% RSLogix 500 project HotWater_HX_12032008.RSS, saved by version 8.10.00.24 %
PROJECT "B8_HW"    % processor: Bul.1763 MicroLogix 1100 Series A %

PROGRAM FILES
  LAD 2 "MAIN"  10 rungs
  LAD 4 "ANALOG IN"  10 rungs
  LAD 5 "PUMP 3"  17 rungs
  LAD 6 "PUMP 4"  16 rungs
  LAD 7 "PRESS PID"  15 rungs
  LAD 8 "TEMP PID"  16 rungs
  LAD 9 "ANALOG OUT"  8 rungs
  LAD 10 "LCD INFO"  13 rungs

DATA FILES
  O0 OUTPUT  8 elements
  I1 INPUT  22 elements
  S2 STATUS  66 elements
  B3 BINARY  11 elements
  T4 TIMER  57 elements
  C5 COUNTER  10 elements
  R6 CONTROL  1 elements
  N7 INTEGER  100 elements
  F8 FLOAT  1 elements
  PD9   12 elements
  N10   200 elements
  N11   52 elements
  N12   40 elements
  F13   40 elements

LADDER 2 "MAIN"
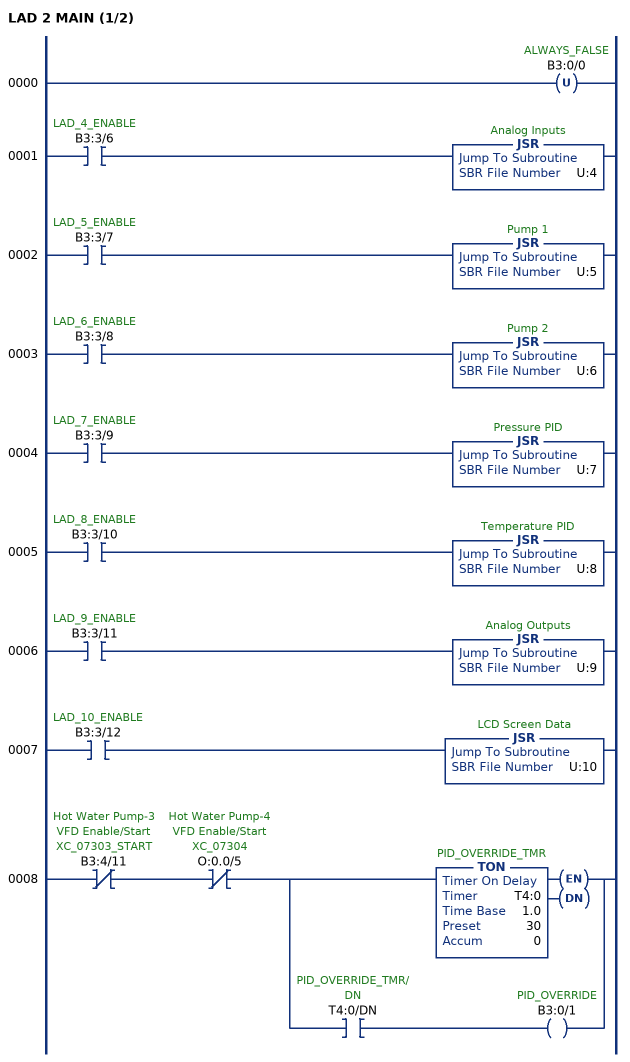
% Rung: 0 %
SOR OTU B3:0/0 EOR
%   B3:0/0  ALWAYS_FALSE %
% Rung: 1 %
SOR XIC B3:3/6 JSR U:4 EOR
%   B3:3/6  LAD_4_ENABLE %
%   U:4  "Analog Inputs" %
% Rung: 2 %
SOR XIC B3:3/7 JSR U:5 EOR
%   B3:3/7  LAD_5_ENABLE %
%   U:5  "Pump 1" %
% Rung: 3 %
SOR XIC B3:3/8 JSR U:6 EOR
%   B3:3/8  LAD_6_ENABLE %
%   U:6  "Pump 2" %
% Rung: 4 %
SOR XIC B3:3/9 JSR U:7 EOR
%   B3:3/9  LAD_7_ENABLE %
%   U:7  "Pressure PID" %
% Rung: 5 %
SOR XIC B3:3/10 JSR U:8 EOR
%   B3:3/10  LAD_8_ENABLE %
%   U:8  "Temperature PID" %
% Rung: 6 %
SOR XIC B3:3/11 JSR U:9 EOR
%   B3:3/11  LAD_9_ENABLE %
%   U:9  "Analog Outputs" %
% Rung: 7 %
SOR XIC B3:3/12 JSR U:10 EOR
%   B3:3/12  LAD_10_ENABLE %
%   U:10  "LCD Screen Data" %
% Rung: 8 %
SOR XIO B3:4/11 XIO O:0.0/5 BST TON T4:0 1.0 30 0 NXB XIC T4:0/DN OTE B3:0/1 BND EOR
%   B3:4/11  XC_07303_START  "Hot Water Pump-3 VFD Enable/Start" %
%   O:0.0/5  XC_07304  "Hot Water Pump-4 VFD Enable/Start" %
%   T4:0  PID_OVERRIDE_TMR %
%   B3:0/1  PID_OVERRIDE %

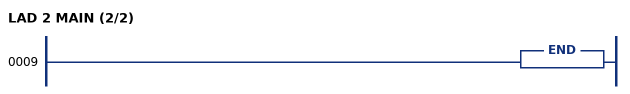
% Rung: 9 %
SOR END EOR

LADDER 4 "ANALOG IN"
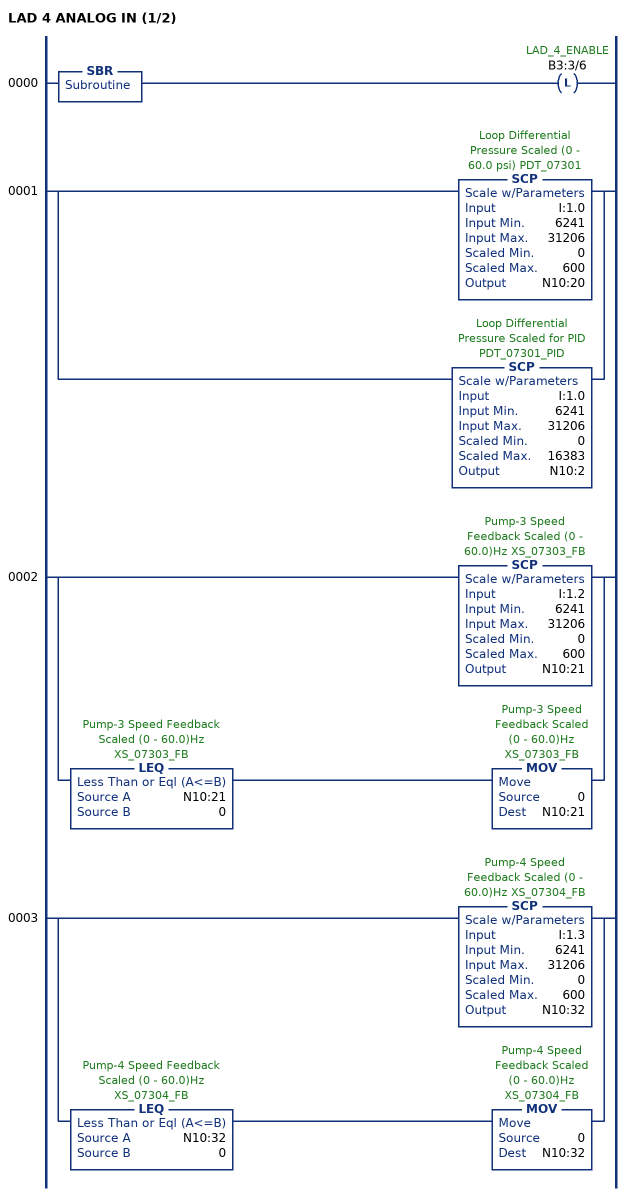
% Rung: 0 %
SOR SBR OTL B3:3/6 EOR
%   B3:3/6  LAD_4_ENABLE %
% Rung: 1 %
SOR BST SCP I:1.0 6241 31206 0 600 N10:20 NXB SCP I:1.0 6241 31206 0 16383 N10:2 BND EOR
%   I:1.0  PDT_07301_RAW  "Loop Differential Pressure Scaled (0.0 - 60.0) psi" %
%   N10:20  PDT_07301  "Loop Differential Pressure Scaled (0 - 60.0 psi)" %
%   N10:2  PDT_07301_PID  "Loop Differential Pressure Scaled for PID" %
% Rung: 2 %
SOR BST SCP I:1.2 6241 31206 0 600 N10:21 NXB LEQ N10:21 0 MOV 0 N10:21 BND EOR
%   I:1.2  XS_07303_FB_RAW  "Pump-3 VFD Speed Feedback" %
%   N10:21  XS_07303_FB  "Pump-3 Speed Feedback Scaled (0 - 60.0)Hz" %
% Rung: 3 %
SOR BST SCP I:1.3 6241 31206 0 600 N10:32 NXB LEQ N10:32 0 MOV 0 N10:32 BND EOR
%   I:1.3  XS_07304_FB_RAW  "Pump-4 VFD Speed Feedback" %
%   N10:32  XS_07304_FB  "Pump-4 Speed Feedback Scaled (0 - 60.0)Hz" %

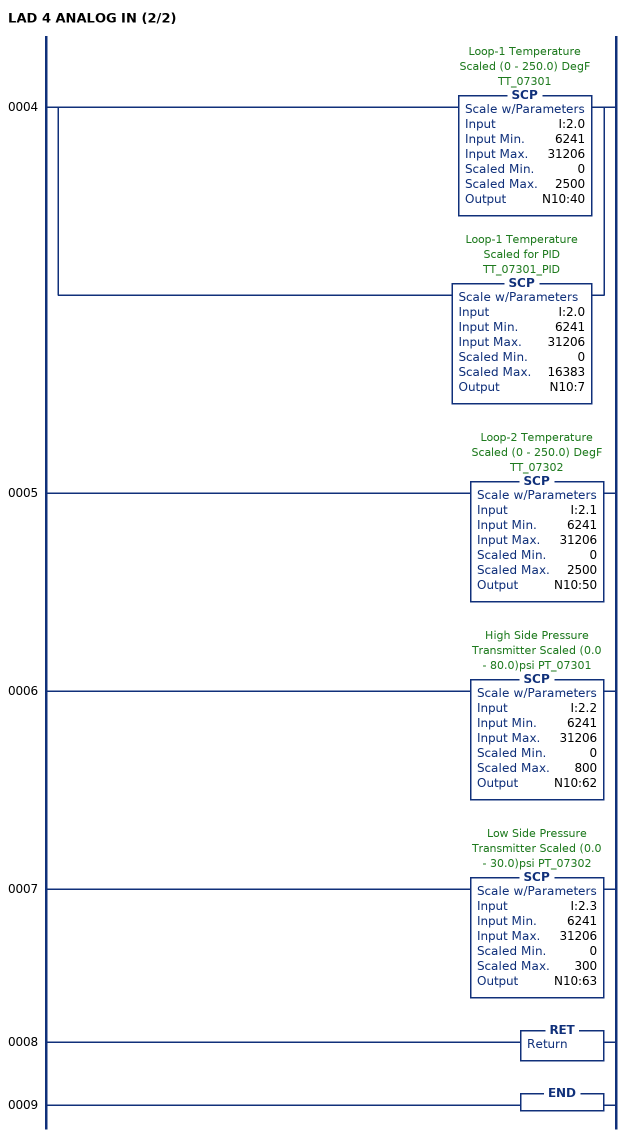
% Rung: 4 %
SOR BST SCP I:2.0 6241 31206 0 2500 N10:40 NXB SCP I:2.0 6241 31206 0 16383 N10:7 BND EOR
%   I:2.0  TT_07301_RAW  "Loop-1 Temperature Transmitter Scaled (0 - 250.0) DegF" %
%   N10:40  TT_07301  "Loop-1 Temperature Scaled (0 - 250.0) DegF" %
%   N10:7  TT_07301_PID  "Loop-1 Temperature Scaled for PID" %
% Rung: 5 %
SOR SCP I:2.1 6241 31206 0 2500 N10:50 EOR
%   I:2.1  TT_07302_RAW  "Loop-2 Temperature Transmitter Scaled (0 - 250.0) DegF" %
%   N10:50  TT_07302  "Loop-2 Temperature Scaled (0 - 250.0) DegF" %
% Rung: 6 %
SOR SCP I:2.2 6241 31206 0 800 N10:62 EOR
%   I:2.2  PT_07301_RAW  "High Side Pressure Transmitter Scaled (0.0 - 80.0)psi" %
%   N10:62  PT_07301  "High Side Pressure Transmitter Scaled (0.0 - 80.0)psi" %
% Rung: 7 %
SOR SCP I:2.3 6241 31206 0 300 N10:63 EOR
%   I:2.3  PT_07302_RAW  "Low Side Pressure Transmitter Scaled (0.0 - 30.0)psi" %
%   N10:63  PT_07302  "Low Side Pressure Transmitter Scaled (0.0 - 30.0)psi" %
% Rung: 8 %
SOR RET EOR
% Rung: 9 %
SOR END EOR

LADDER 5 "PUMP 3"
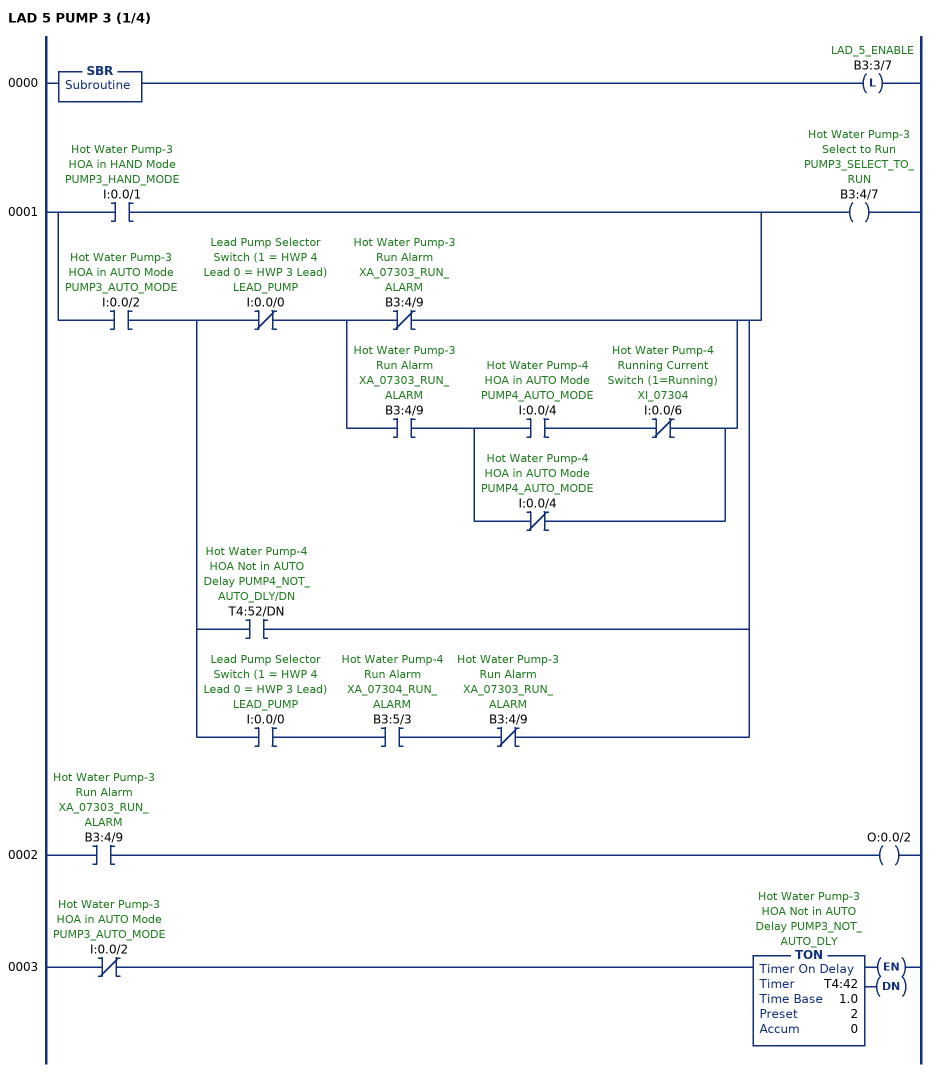
% Rung: 0 %
SOR SBR OTL B3:3/7 EOR
%   B3:3/7  LAD_5_ENABLE %
% Rung: 1 %
SOR BST XIC I:0.0/1 NXB XIC I:0.0/2 BST XIO I:0.0/0 BST XIO B3:4/9 NXB XIC B3:4/9 BST XIC I:0.0/4 XIO I:0.0/6 NXB XIO I:0.0/4 BND BND NXB XIC T4:52/DN NXB XIC I:0.0/0 XIC B3:5/3 XIO B3:4/9 BND BND OTE B3:4/7 EOR
%   I:0.0/1  PUMP3_HAND_MODE  "Hot Water Pump-3 HOA in HAND Mode" %
%   I:0.0/2  PUMP3_AUTO_MODE  "Hot Water Pump-3 HOA in AUTO Mode" %
%   I:0.0/0  LEAD_PUMP  "Lead Pump Selector Switch (1 = HWP 4 Lead 0 = HWP 3 Lead)" %
%   B3:4/9  XA_07303_RUN_ALARM  "Hot Water Pump-3 Run Alarm" %
%   I:0.0/4  PUMP4_AUTO_MODE  "Hot Water Pump-4 HOA in AUTO Mode" %
%   I:0.0/6  XI_07304  "Hot Water Pump-4 Running Current Switch (1=Running)" %
%   T4:52  PUMP4_NOT_AUTO_DLY  "Hot Water Pump-4 HOA Not in AUTO Delay" %
%   B3:5/3  XA_07304_RUN_ALARM  "Hot Water Pump-4 Run Alarm" %
%   B3:4/7  PUMP3_SELECT_TO_RUN  "Hot Water Pump-3 Select to Run" %
% Rung: 2 %
SOR XIC B3:4/9 OTE O:0.0/2 EOR
%   B3:4/9  XA_07303_RUN_ALARM  "Hot Water Pump-3 Run Alarm" %
% Rung: 3 %
SOR XIO I:0.0/2 TON T4:42 1.0 2 0 EOR
%   I:0.0/2  PUMP3_AUTO_MODE  "Hot Water Pump-3 HOA in AUTO Mode" %
%   T4:42  PUMP3_NOT_AUTO_DLY  "Hot Water Pump-3 HOA Not in AUTO Delay" %

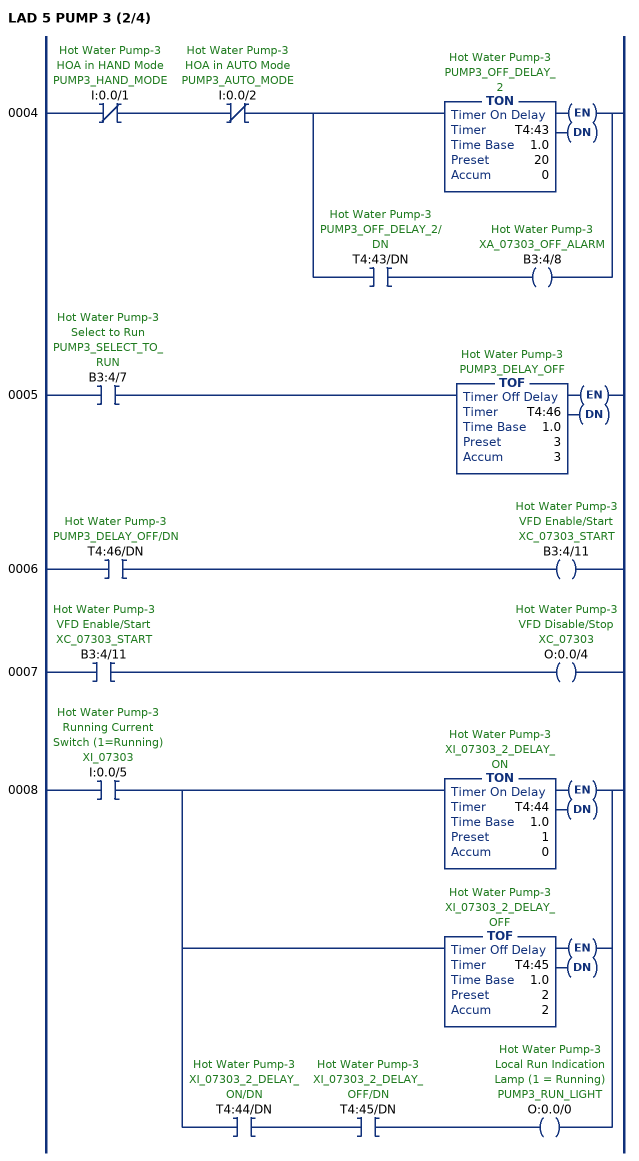
% Rung: 4 %
SOR XIO I:0.0/1 XIO I:0.0/2 BST TON T4:43 1.0 20 0 NXB XIC T4:43/DN OTE B3:4/8 BND EOR
%   I:0.0/1  PUMP3_HAND_MODE  "Hot Water Pump-3 HOA in HAND Mode" %
%   I:0.0/2  PUMP3_AUTO_MODE  "Hot Water Pump-3 HOA in AUTO Mode" %
%   T4:43  PUMP3_OFF_DELAY_2  "Hot Water Pump-3" %
%   B3:4/8  XA_07303_OFF_ALARM  "Hot Water Pump-3" %
% Rung: 5 %
SOR XIC B3:4/7 TOF T4:46 1.0 3 3 EOR
%   B3:4/7  PUMP3_SELECT_TO_RUN  "Hot Water Pump-3 Select to Run" %
%   T4:46  PUMP3_DELAY_OFF  "Hot Water Pump-3" %
% Rung: 6 %
SOR XIC T4:46/DN OTE B3:4/11 EOR
%   T4:46  PUMP3_DELAY_OFF  "Hot Water Pump-3" %
%   B3:4/11  XC_07303_START  "Hot Water Pump-3 VFD Enable/Start" %
% Rung: 7 %
SOR XIC B3:4/11 OTE O:0.0/4 EOR
%   B3:4/11  XC_07303_START  "Hot Water Pump-3 VFD Enable/Start" %
%   O:0.0/4  XC_07303  "Hot Water Pump-3 VFD Disable/Stop" %
% Rung: 8 %
SOR XIC I:0.0/5 BST TON T4:44 1.0 1 0 NXB TOF T4:45 1.0 2 2 NXB XIC T4:44/DN XIC T4:45/DN OTE O:0.0/0 BND EOR
%   I:0.0/5  XI_07303  "Hot Water Pump-3 Running Current Switch (1=Running)" %
%   T4:44  XI_07303_2_DELAY_ON  "Hot Water Pump-3" %
%   T4:45  XI_07303_2_DELAY_OFF  "Hot Water Pump-3" %
%   O:0.0/0  PUMP3_RUN_LIGHT  "Hot Water Pump-3 Local Run Indication Lamp (1 = Running)" %

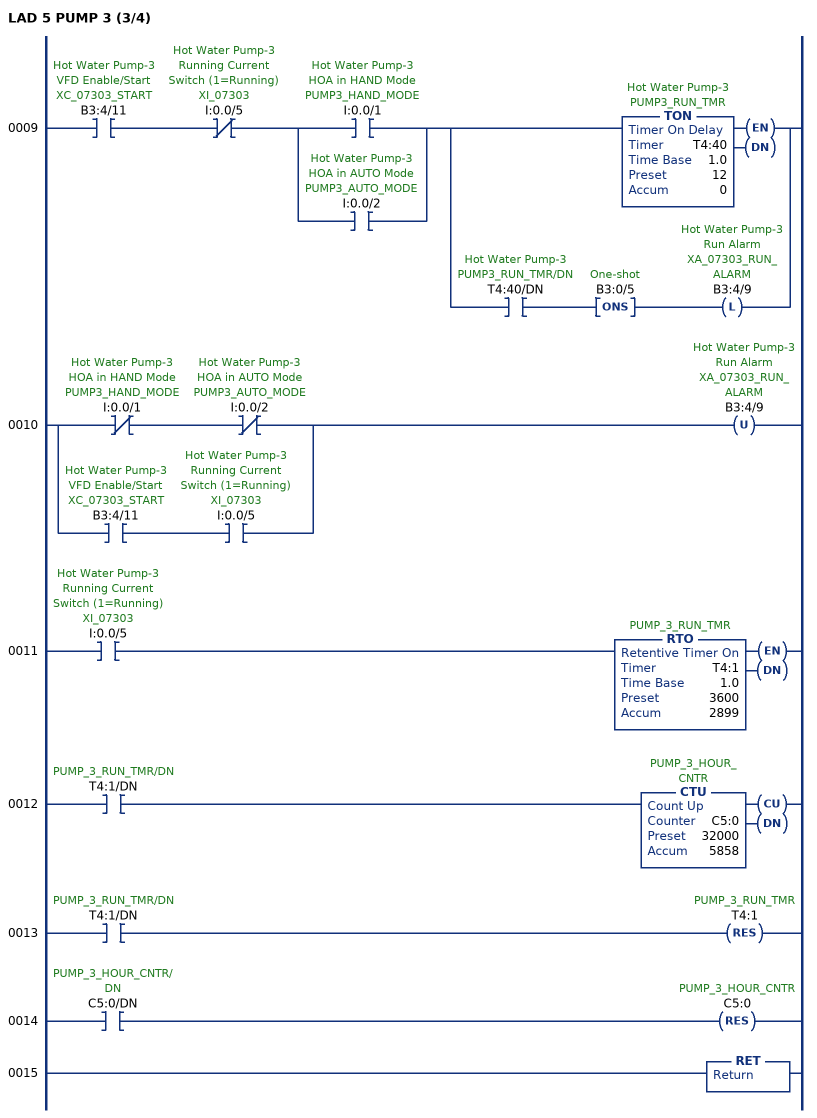
% Rung: 9 %
SOR XIC B3:4/11 XIO I:0.0/5 BST XIC I:0.0/1 NXB XIC I:0.0/2 BND BST TON T4:40 1.0 12 0 NXB XIC T4:40/DN ONS B3:0/5 OTL B3:4/9 BND EOR
%   B3:4/11  XC_07303_START  "Hot Water Pump-3 VFD Enable/Start" %
%   I:0.0/5  XI_07303  "Hot Water Pump-3 Running Current Switch (1=Running)" %
%   I:0.0/1  PUMP3_HAND_MODE  "Hot Water Pump-3 HOA in HAND Mode" %
%   I:0.0/2  PUMP3_AUTO_MODE  "Hot Water Pump-3 HOA in AUTO Mode" %
%   T4:40  PUMP3_RUN_TMR  "Hot Water Pump-3" %
%   B3:0/5  "One-shot" %
%   B3:4/9  XA_07303_RUN_ALARM  "Hot Water Pump-3 Run Alarm" %
% Rung: 10 %
SOR BST XIO I:0.0/1 XIO I:0.0/2 NXB XIC B3:4/11 XIC I:0.0/5 BND OTU B3:4/9 EOR
%   I:0.0/1  PUMP3_HAND_MODE  "Hot Water Pump-3 HOA in HAND Mode" %
%   I:0.0/2  PUMP3_AUTO_MODE  "Hot Water Pump-3 HOA in AUTO Mode" %
%   B3:4/11  XC_07303_START  "Hot Water Pump-3 VFD Enable/Start" %
%   I:0.0/5  XI_07303  "Hot Water Pump-3 Running Current Switch (1=Running)" %
%   B3:4/9  XA_07303_RUN_ALARM  "Hot Water Pump-3 Run Alarm" %
% Rung: 11 %
SOR XIC I:0.0/5 RTO T4:1 1.0 3600 2899 EOR
%   I:0.0/5  XI_07303  "Hot Water Pump-3 Running Current Switch (1=Running)" %
%   T4:1  PUMP_3_RUN_TMR %
% Rung: 12 %
SOR XIC T4:1/DN CTU C5:0 32000 5858 EOR
%   T4:1  PUMP_3_RUN_TMR %
%   C5:0  PUMP_3_HOUR_CNTR %
% Rung: 13 %
SOR XIC T4:1/DN RES T4:1 EOR
%   T4:1  PUMP_3_RUN_TMR %
% Rung: 14 %
SOR XIC C5:0/DN RES C5:0 EOR
%   C5:0  PUMP_3_HOUR_CNTR %
% Rung: 15 %
SOR RET EOR

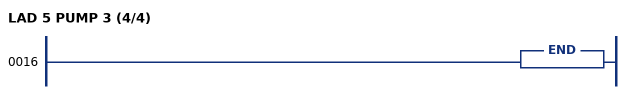
% Rung: 16 %
SOR END EOR

LADDER 6 "PUMP 4"
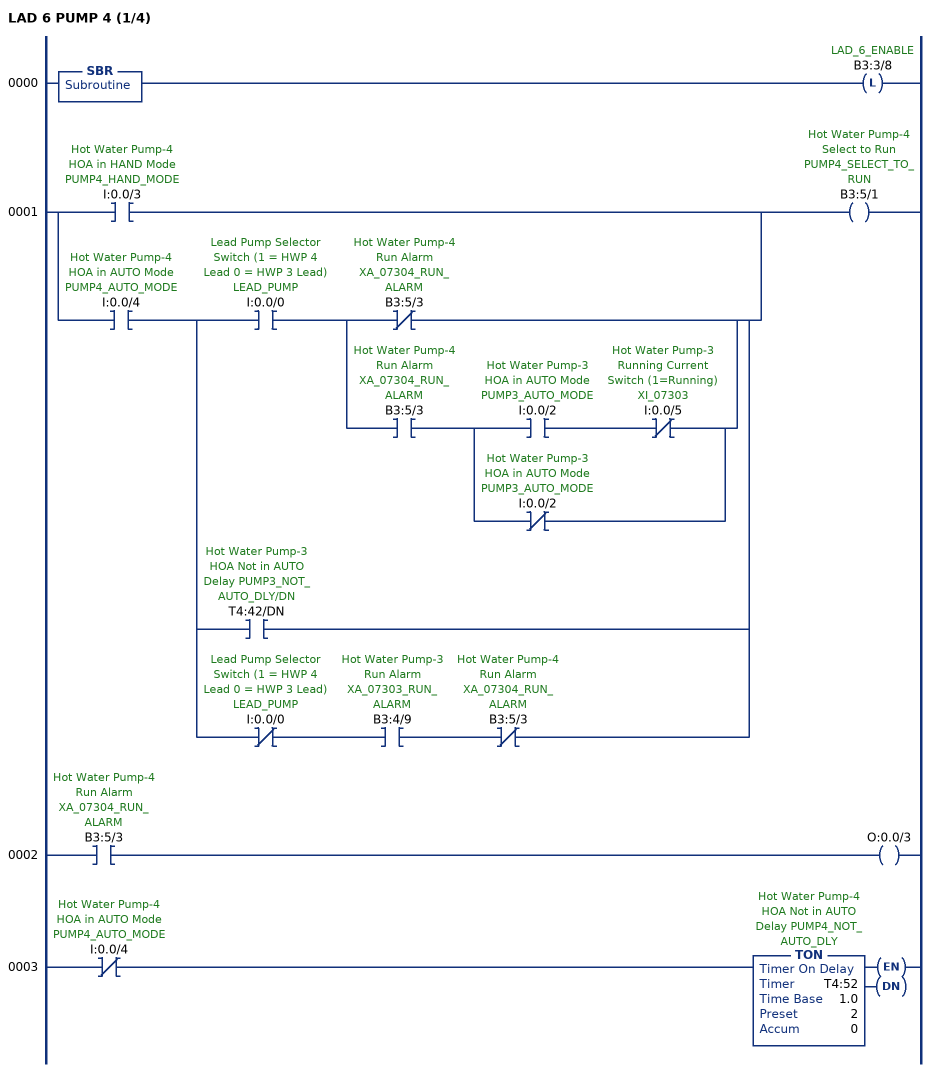
% Rung: 0 %
SOR SBR OTL B3:3/8 EOR
%   B3:3/8  LAD_6_ENABLE %
% Rung: 1 %
SOR BST XIC I:0.0/3 NXB XIC I:0.0/4 BST XIC I:0.0/0 BST XIO B3:5/3 NXB XIC B3:5/3 BST XIC I:0.0/2 XIO I:0.0/5 NXB XIO I:0.0/2 BND BND NXB XIC T4:42/DN NXB XIO I:0.0/0 XIC B3:4/9 XIO B3:5/3 BND BND OTE B3:5/1 EOR
%   I:0.0/3  PUMP4_HAND_MODE  "Hot Water Pump-4 HOA in HAND Mode" %
%   I:0.0/4  PUMP4_AUTO_MODE  "Hot Water Pump-4 HOA in AUTO Mode" %
%   I:0.0/0  LEAD_PUMP  "Lead Pump Selector Switch (1 = HWP 4 Lead 0 = HWP 3 Lead)" %
%   B3:5/3  XA_07304_RUN_ALARM  "Hot Water Pump-4 Run Alarm" %
%   I:0.0/2  PUMP3_AUTO_MODE  "Hot Water Pump-3 HOA in AUTO Mode" %
%   I:0.0/5  XI_07303  "Hot Water Pump-3 Running Current Switch (1=Running)" %
%   T4:42  PUMP3_NOT_AUTO_DLY  "Hot Water Pump-3 HOA Not in AUTO Delay" %
%   B3:4/9  XA_07303_RUN_ALARM  "Hot Water Pump-3 Run Alarm" %
%   B3:5/1  PUMP4_SELECT_TO_RUN  "Hot Water Pump-4 Select to Run" %
% Rung: 2 %
SOR XIC B3:5/3 OTE O:0.0/3 EOR
%   B3:5/3  XA_07304_RUN_ALARM  "Hot Water Pump-4 Run Alarm" %
% Rung: 3 %
SOR XIO I:0.0/4 TON T4:52 1.0 2 0 EOR
%   I:0.0/4  PUMP4_AUTO_MODE  "Hot Water Pump-4 HOA in AUTO Mode" %
%   T4:52  PUMP4_NOT_AUTO_DLY  "Hot Water Pump-4 HOA Not in AUTO Delay" %

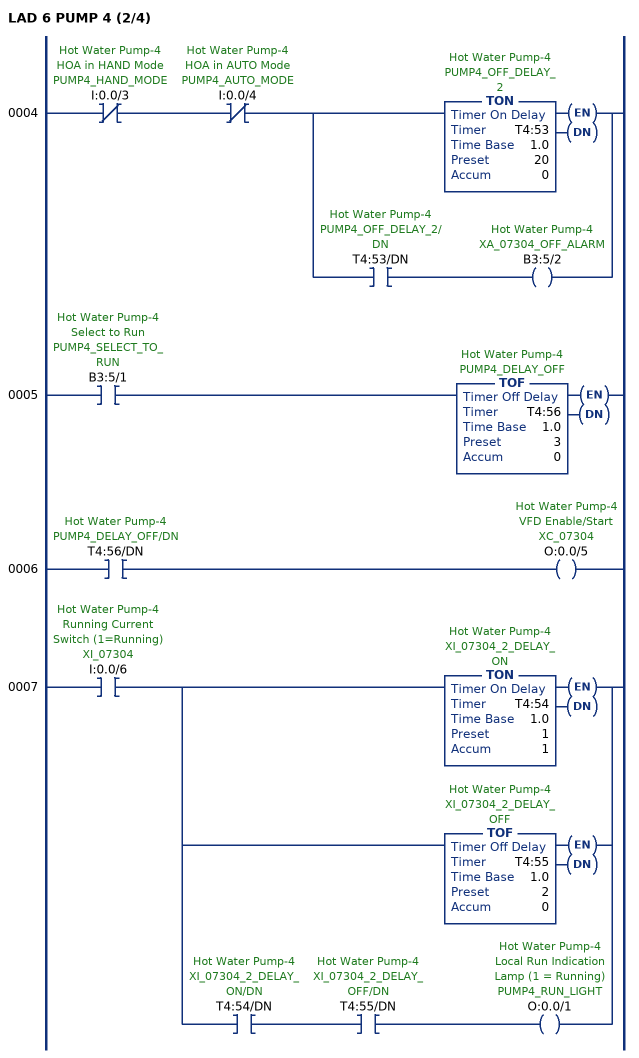
% Rung: 4 %
SOR XIO I:0.0/3 XIO I:0.0/4 BST TON T4:53 1.0 20 0 NXB XIC T4:53/DN OTE B3:5/2 BND EOR
%   I:0.0/3  PUMP4_HAND_MODE  "Hot Water Pump-4 HOA in HAND Mode" %
%   I:0.0/4  PUMP4_AUTO_MODE  "Hot Water Pump-4 HOA in AUTO Mode" %
%   T4:53  PUMP4_OFF_DELAY_2  "Hot Water Pump-4" %
%   B3:5/2  XA_07304_OFF_ALARM  "Hot Water Pump-4" %
% Rung: 5 %
SOR XIC B3:5/1 TOF T4:56 1.0 3 0 EOR
%   B3:5/1  PUMP4_SELECT_TO_RUN  "Hot Water Pump-4 Select to Run" %
%   T4:56  PUMP4_DELAY_OFF  "Hot Water Pump-4" %
% Rung: 6 %
SOR XIC T4:56/DN OTE O:0.0/5 EOR
%   T4:56  PUMP4_DELAY_OFF  "Hot Water Pump-4" %
%   O:0.0/5  XC_07304  "Hot Water Pump-4 VFD Enable/Start" %
% Rung: 7 %
SOR XIC I:0.0/6 BST TON T4:54 1.0 1 1 NXB TOF T4:55 1.0 2 0 NXB XIC T4:54/DN XIC T4:55/DN OTE O:0.0/1 BND EOR
%   I:0.0/6  XI_07304  "Hot Water Pump-4 Running Current Switch (1=Running)" %
%   T4:54  XI_07304_2_DELAY_ON  "Hot Water Pump-4" %
%   T4:55  XI_07304_2_DELAY_OFF  "Hot Water Pump-4" %
%   O:0.0/1  PUMP4_RUN_LIGHT  "Hot Water Pump-4 Local Run Indication Lamp (1 = Running)" %

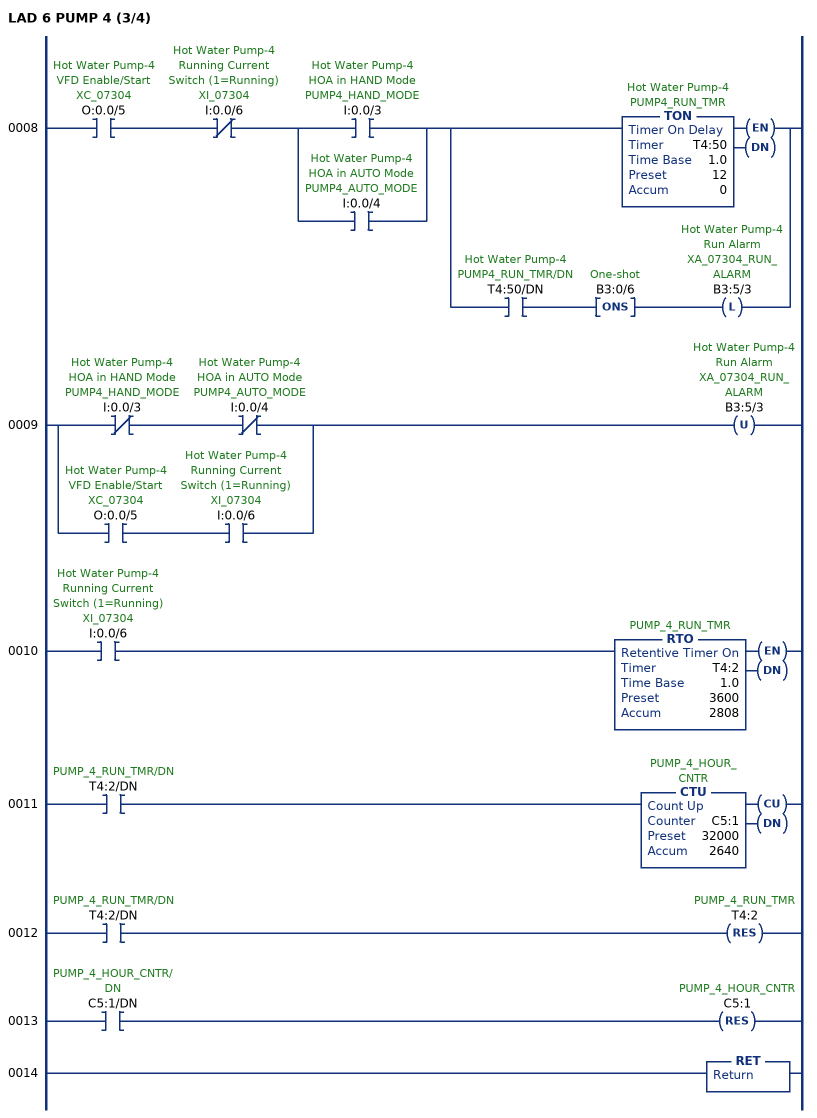
% Rung: 8 %
SOR XIC O:0.0/5 XIO I:0.0/6 BST XIC I:0.0/3 NXB XIC I:0.0/4 BND BST TON T4:50 1.0 12 0 NXB XIC T4:50/DN ONS B3:0/6 OTL B3:5/3 BND EOR
%   O:0.0/5  XC_07304  "Hot Water Pump-4 VFD Enable/Start" %
%   I:0.0/6  XI_07304  "Hot Water Pump-4 Running Current Switch (1=Running)" %
%   I:0.0/3  PUMP4_HAND_MODE  "Hot Water Pump-4 HOA in HAND Mode" %
%   I:0.0/4  PUMP4_AUTO_MODE  "Hot Water Pump-4 HOA in AUTO Mode" %
%   T4:50  PUMP4_RUN_TMR  "Hot Water Pump-4" %
%   B3:0/6  "One-shot" %
%   B3:5/3  XA_07304_RUN_ALARM  "Hot Water Pump-4 Run Alarm" %
% Rung: 9 %
SOR BST XIO I:0.0/3 XIO I:0.0/4 NXB XIC O:0.0/5 XIC I:0.0/6 BND OTU B3:5/3 EOR
%   I:0.0/3  PUMP4_HAND_MODE  "Hot Water Pump-4 HOA in HAND Mode" %
%   I:0.0/4  PUMP4_AUTO_MODE  "Hot Water Pump-4 HOA in AUTO Mode" %
%   O:0.0/5  XC_07304  "Hot Water Pump-4 VFD Enable/Start" %
%   I:0.0/6  XI_07304  "Hot Water Pump-4 Running Current Switch (1=Running)" %
%   B3:5/3  XA_07304_RUN_ALARM  "Hot Water Pump-4 Run Alarm" %
% Rung: 10 %
SOR XIC I:0.0/6 RTO T4:2 1.0 3600 2808 EOR
%   I:0.0/6  XI_07304  "Hot Water Pump-4 Running Current Switch (1=Running)" %
%   T4:2  PUMP_4_RUN_TMR %
% Rung: 11 %
SOR XIC T4:2/DN CTU C5:1 32000 2640 EOR
%   T4:2  PUMP_4_RUN_TMR %
%   C5:1  PUMP_4_HOUR_CNTR %
% Rung: 12 %
SOR XIC T4:2/DN RES T4:2 EOR
%   T4:2  PUMP_4_RUN_TMR %
% Rung: 13 %
SOR XIC C5:1/DN RES C5:1 EOR
%   C5:1  PUMP_4_HOUR_CNTR %
% Rung: 14 %
SOR RET EOR

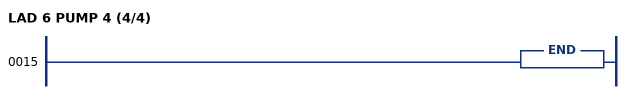
% Rung: 15 %
SOR END EOR

LADDER 7 "PRESS PID"
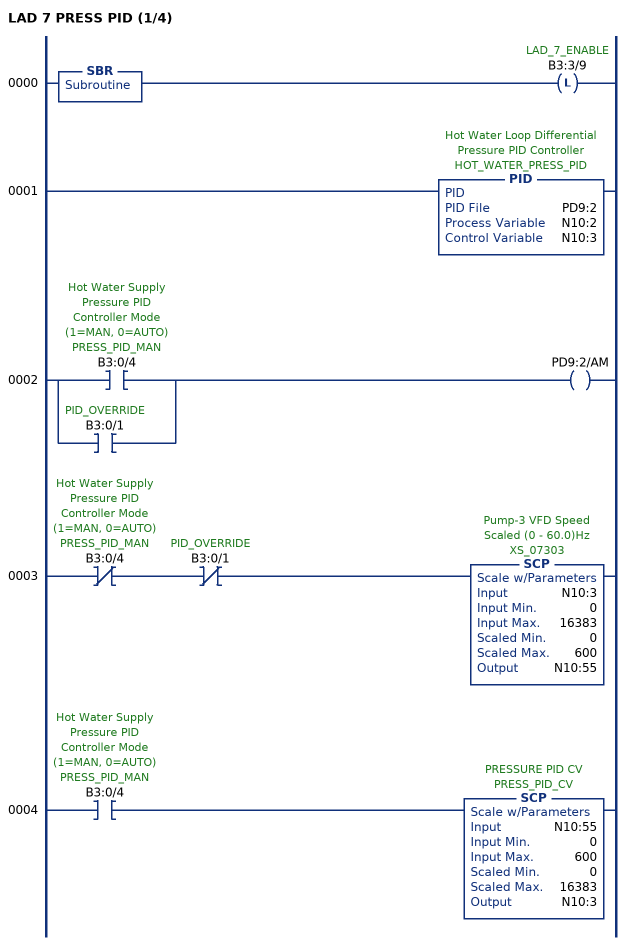
% Rung: 0 %
SOR SBR OTL B3:3/9 EOR
%   B3:3/9  LAD_7_ENABLE %
% Rung: 1 %
SOR PID PD9:2 N10:2 N10:3 EOR
%   PD9:2  HOT_WATER_PRESS_PID  "Hot Water Loop Differential Pressure PID Controller" %
%   N10:2  PDT_07301_PID  "Loop Differential Pressure Scaled for PID" %
%   N10:3  PRESS_PID_CV  "PRESSURE PID CV" %
% Rung: 2 %
SOR BST XIC B3:0/4 NXB XIC B3:0/1 BND OTE PD9:2/AM EOR
%   B3:0/4  PRESS_PID_MAN  "Hot Water Supply Pressure PID Controller Mode (1=MAN, 0=AUTO)" %
%   B3:0/1  PID_OVERRIDE %
% Rung: 3 %
SOR XIO B3:0/4 XIO B3:0/1 SCP N10:3 0 16383 0 600 N10:55 EOR
%   B3:0/4  PRESS_PID_MAN  "Hot Water Supply Pressure PID Controller Mode (1=MAN, 0=AUTO)" %
%   B3:0/1  PID_OVERRIDE %
%   N10:3  PRESS_PID_CV  "PRESSURE PID CV" %
%   N10:55  XS_07303  "Pump-3 VFD Speed Scaled (0 - 60.0)Hz" %
% Rung: 4 %
SOR XIC B3:0/4 SCP N10:55 0 600 0 16383 N10:3 EOR
%   B3:0/4  PRESS_PID_MAN  "Hot Water Supply Pressure PID Controller Mode (1=MAN, 0=AUTO)" %
%   N10:55  XS_07303  "Pump-3 VFD Speed Scaled (0 - 60.0)Hz" %
%   N10:3  PRESS_PID_CV  "PRESSURE PID CV" %

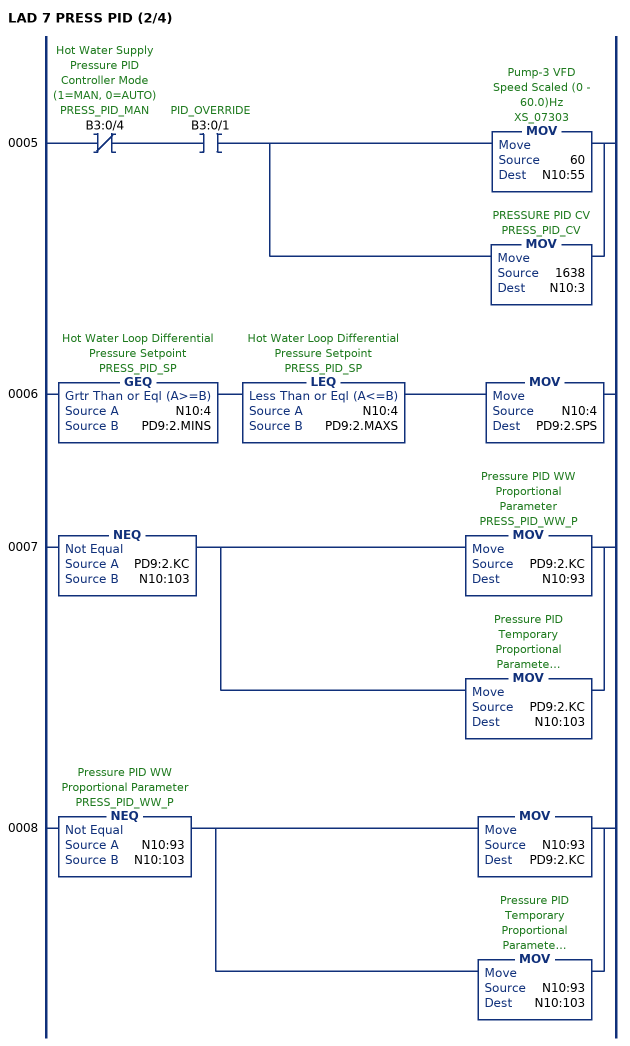
% Rung: 5 %
SOR XIO B3:0/4 XIC B3:0/1 BST MOV 60 N10:55 NXB MOV 1638 N10:3 BND EOR
%   B3:0/4  PRESS_PID_MAN  "Hot Water Supply Pressure PID Controller Mode (1=MAN, 0=AUTO)" %
%   B3:0/1  PID_OVERRIDE %
%   N10:55  XS_07303  "Pump-3 VFD Speed Scaled (0 - 60.0)Hz" %
%   N10:3  PRESS_PID_CV  "PRESSURE PID CV" %
% Rung: 6 %
SOR GEQ N10:4 PD9:2.MINS LEQ N10:4 PD9:2.MAXS MOV N10:4 PD9:2.SPS EOR
%   N10:4  PRESS_PID_SP  "Hot Water Loop Differential Pressure Setpoint" %
% Rung: 7 %
SOR NEQ PD9:2.KC N10:103 BST MOV PD9:2.KC N10:93 NXB MOV PD9:2.KC N10:103 BND EOR
%   N10:103  PRESS_PID_WW_TMP_P  "Pressure PID Temporary Proportional Parameter" %
%   N10:93  PRESS_PID_WW_P  "Pressure PID WW Proportional Parameter" %
% Rung: 8 %
SOR NEQ N10:93 N10:103 BST MOV N10:93 PD9:2.KC NXB MOV N10:93 N10:103 BND EOR
%   N10:93  PRESS_PID_WW_P  "Pressure PID WW Proportional Parameter" %
%   N10:103  PRESS_PID_WW_TMP_P  "Pressure PID Temporary Proportional Parameter" %

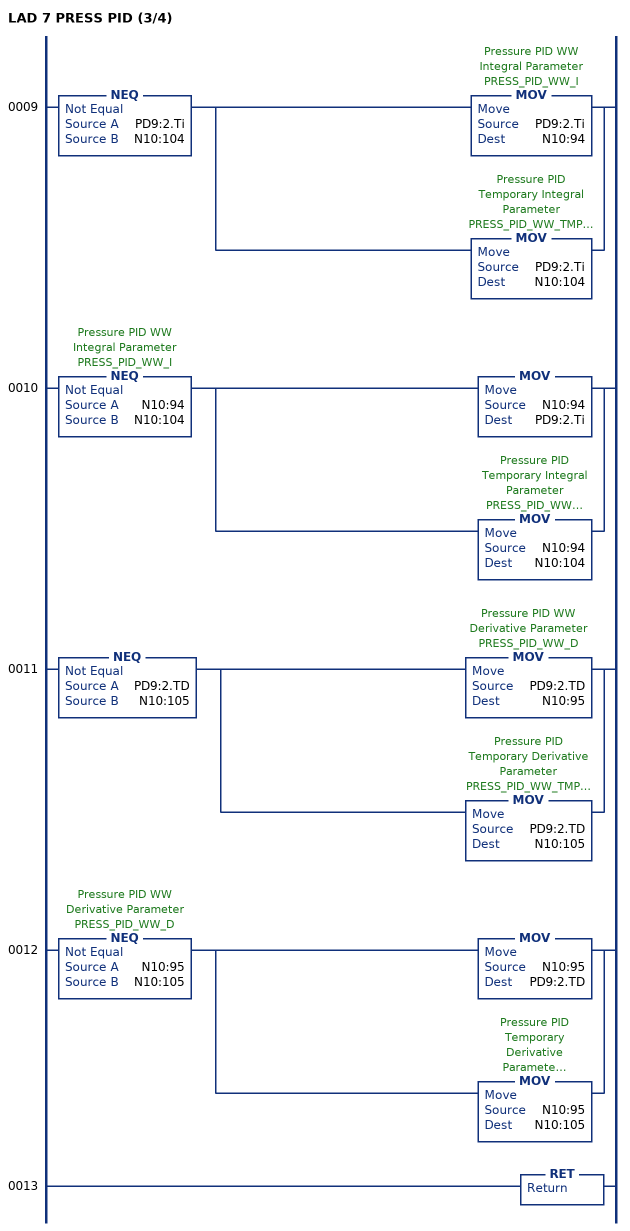
% Rung: 9 %
SOR NEQ PD9:2.Ti N10:104 BST MOV PD9:2.Ti N10:94 NXB MOV PD9:2.Ti N10:104 BND EOR
%   N10:104  PRESS_PID_WW_TMP_I  "Pressure PID Temporary Integral Parameter" %
%   N10:94  PRESS_PID_WW_I  "Pressure PID WW Integral Parameter" %
% Rung: 10 %
SOR NEQ N10:94 N10:104 BST MOV N10:94 PD9:2.Ti NXB MOV N10:94 N10:104 BND EOR
%   N10:94  PRESS_PID_WW_I  "Pressure PID WW Integral Parameter" %
%   N10:104  PRESS_PID_WW_TMP_I  "Pressure PID Temporary Integral Parameter" %
% Rung: 11 %
SOR NEQ PD9:2.TD N10:105 BST MOV PD9:2.TD N10:95 NXB MOV PD9:2.TD N10:105 BND EOR
%   N10:105  PRESS_PID_WW_TMP_D  "Pressure PID Temporary Derivative Parameter" %
%   N10:95  PRESS_PID_WW_D  "Pressure PID WW Derivative Parameter" %
% Rung: 12 %
SOR NEQ N10:95 N10:105 BST MOV N10:95 PD9:2.TD NXB MOV N10:95 N10:105 BND EOR
%   N10:95  PRESS_PID_WW_D  "Pressure PID WW Derivative Parameter" %
%   N10:105  PRESS_PID_WW_TMP_D  "Pressure PID Temporary Derivative Parameter" %
% Rung: 13 %
SOR RET EOR

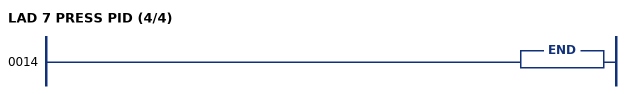
% Rung: 14 %
SOR END EOR

LADDER 8 "TEMP PID"
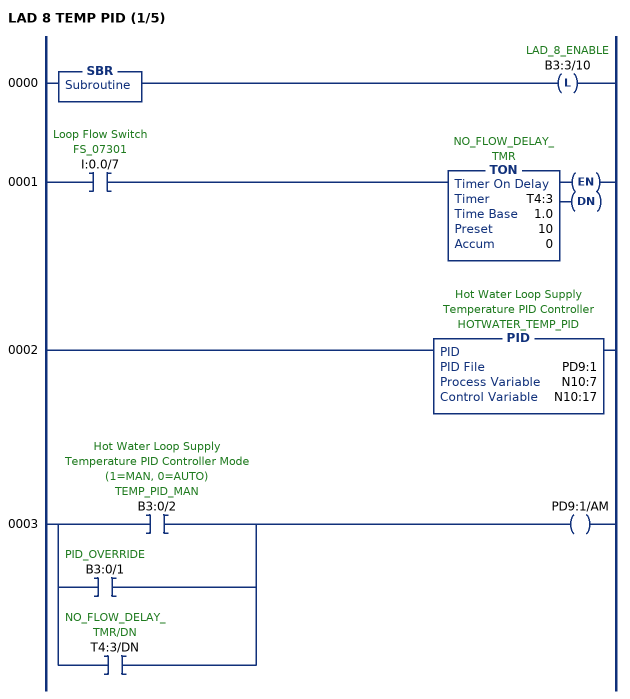
% Rung: 0 %
SOR SBR OTL B3:3/10 EOR
%   B3:3/10  LAD_8_ENABLE %
% Rung: 1 %
SOR XIC I:0.0/7 TON T4:3 1.0 10 0 EOR
%   I:0.0/7  FS_07301  "Loop Flow Switch" %
%   T4:3  NO_FLOW_DELAY_TMR %
% Rung: 2 %
SOR PID PD9:1 N10:7 N10:17 EOR
%   PD9:1  HOTWATER_TEMP_PID  "Hot Water Loop Supply Temperature PID Controller" %
%   N10:7  TT_07301_PID  "Loop-1 Temperature Scaled for PID" %
%   N10:17  TCV_07301_CV  "Hot Water Loop Temperature Control Valve Scaled for PID" %
% Rung: 3 %
SOR BST XIC B3:0/2 NXB XIC B3:0/1 NXB XIC T4:3/DN BND OTE PD9:1/AM EOR
%   B3:0/2  TEMP_PID_MAN  "Hot Water Loop Supply Temperature PID Controller Mode (1=MAN, 0=AUTO)" %
%   B3:0/1  PID_OVERRIDE %
%   T4:3  NO_FLOW_DELAY_TMR %

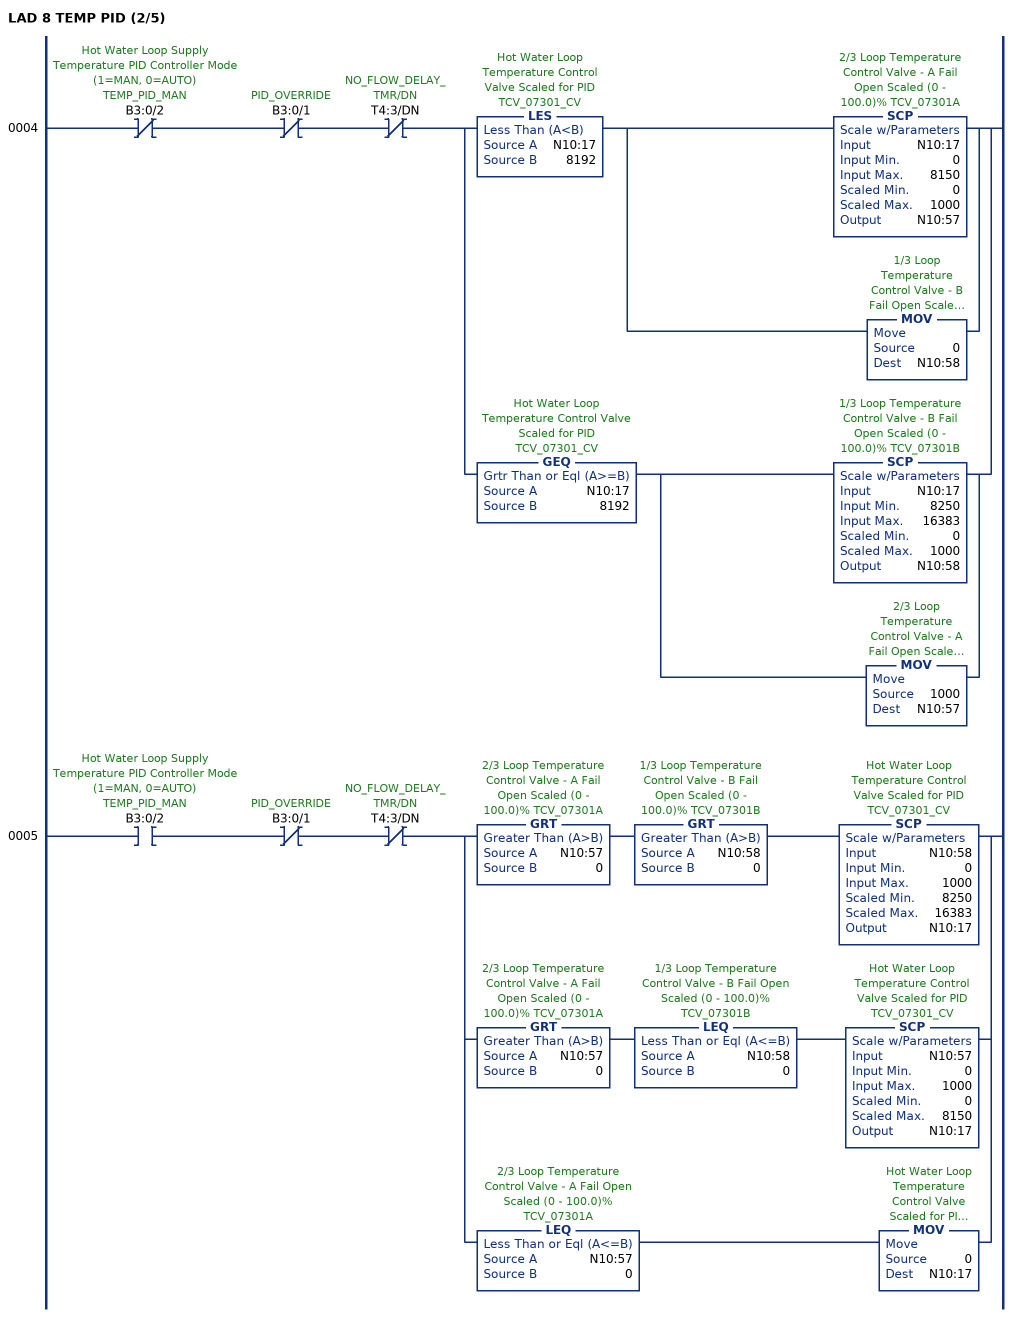
% Rung: 4 %
SOR XIO B3:0/2 XIO B3:0/1 XIO T4:3/DN BST LES N10:17 8192 BST SCP N10:17 0 8150 0 1000 N10:57 NXB MOV 0 N10:58 BND NXB GEQ N10:17 8192 BST SCP N10:17 8250 16383 0 1000 N10:58 NXB MOV 1000 N10:57 BND BND EOR
%   B3:0/2  TEMP_PID_MAN  "Hot Water Loop Supply Temperature PID Controller Mode (1=MAN, 0=AUTO)" %
%   B3:0/1  PID_OVERRIDE %
%   T4:3  NO_FLOW_DELAY_TMR %
%   N10:17  TCV_07301_CV  "Hot Water Loop Temperature Control Valve Scaled for PID" %
%   N10:57  TCV_07301A  "2/3 Loop Temperature Control Valve - A Fail Open Scaled (0 - 100.0)%" %
%   N10:58  TCV_07301B  "1/3 Loop Temperature Control Valve - B Fail Open Scaled (0 - 100.0)%" %
% Rung: 5 %
SOR XIC B3:0/2 XIO B3:0/1 XIO T4:3/DN BST GRT N10:57 0 GRT N10:58 0 SCP N10:58 0 1000 8250 16383 N10:17 NXB GRT N10:57 0 LEQ N10:58 0 SCP N10:57 0 1000 0 8150 N10:17 NXB LEQ N10:57 0 MOV 0 N10:17 BND EOR
%   B3:0/2  TEMP_PID_MAN  "Hot Water Loop Supply Temperature PID Controller Mode (1=MAN, 0=AUTO)" %
%   B3:0/1  PID_OVERRIDE %
%   T4:3  NO_FLOW_DELAY_TMR %
%   N10:57  TCV_07301A  "2/3 Loop Temperature Control Valve - A Fail Open Scaled (0 - 100.0)%" %
%   N10:58  TCV_07301B  "1/3 Loop Temperature Control Valve - B Fail Open Scaled (0 - 100.0)%" %
%   N10:17  TCV_07301_CV  "Hot Water Loop Temperature Control Valve Scaled for PID" %

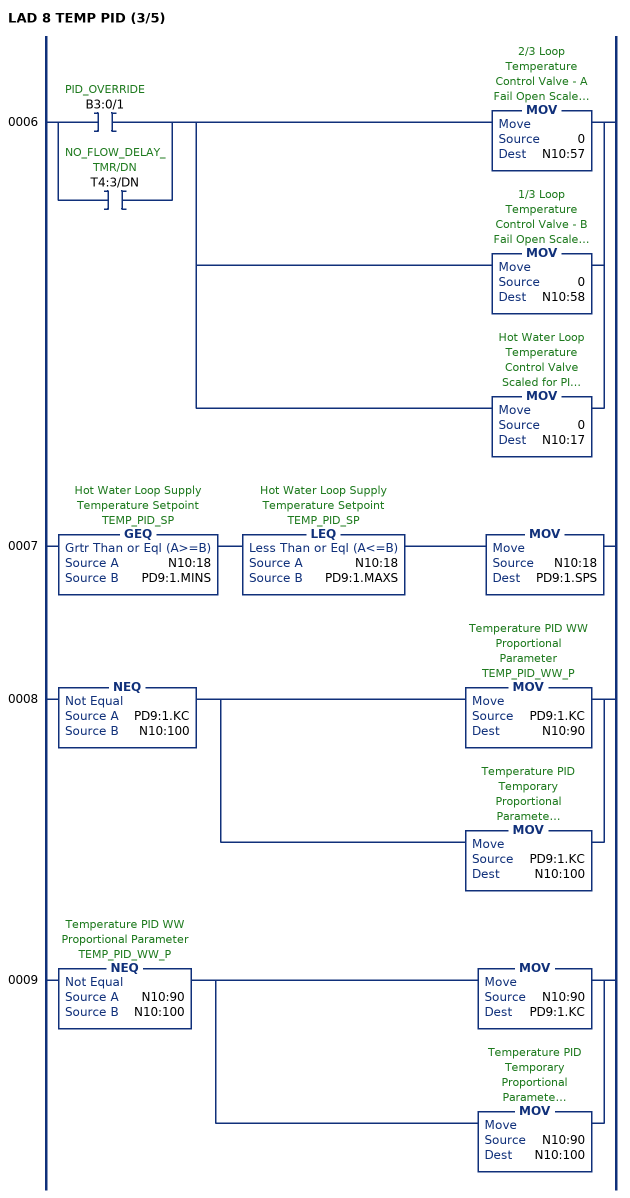
% Rung: 6 %
SOR BST XIC B3:0/1 NXB XIC T4:3/DN BND BST MOV 0 N10:57 NXB MOV 0 N10:58 NXB MOV 0 N10:17 BND EOR
%   B3:0/1  PID_OVERRIDE %
%   T4:3  NO_FLOW_DELAY_TMR %
%   N10:57  TCV_07301A  "2/3 Loop Temperature Control Valve - A Fail Open Scaled (0 - 100.0)%" %
%   N10:58  TCV_07301B  "1/3 Loop Temperature Control Valve - B Fail Open Scaled (0 - 100.0)%" %
%   N10:17  TCV_07301_CV  "Hot Water Loop Temperature Control Valve Scaled for PID" %
% Rung: 7 %
SOR GEQ N10:18 PD9:1.MINS LEQ N10:18 PD9:1.MAXS MOV N10:18 PD9:1.SPS EOR
%   N10:18  TEMP_PID_SP  "Hot Water Loop Supply Temperature Setpoint" %
% Rung: 8 %
SOR NEQ PD9:1.KC N10:100 BST MOV PD9:1.KC N10:90 NXB MOV PD9:1.KC N10:100 BND EOR
%   N10:100  TEMP_PID_WW_TMP_P  "Temperature PID Temporary Proportional Parameter" %
%   N10:90  TEMP_PID_WW_P  "Temperature PID WW Proportional Parameter" %
% Rung: 9 %
SOR NEQ N10:90 N10:100 BST MOV N10:90 PD9:1.KC NXB MOV N10:90 N10:100 BND EOR
%   N10:90  TEMP_PID_WW_P  "Temperature PID WW Proportional Parameter" %
%   N10:100  TEMP_PID_WW_TMP_P  "Temperature PID Temporary Proportional Parameter" %

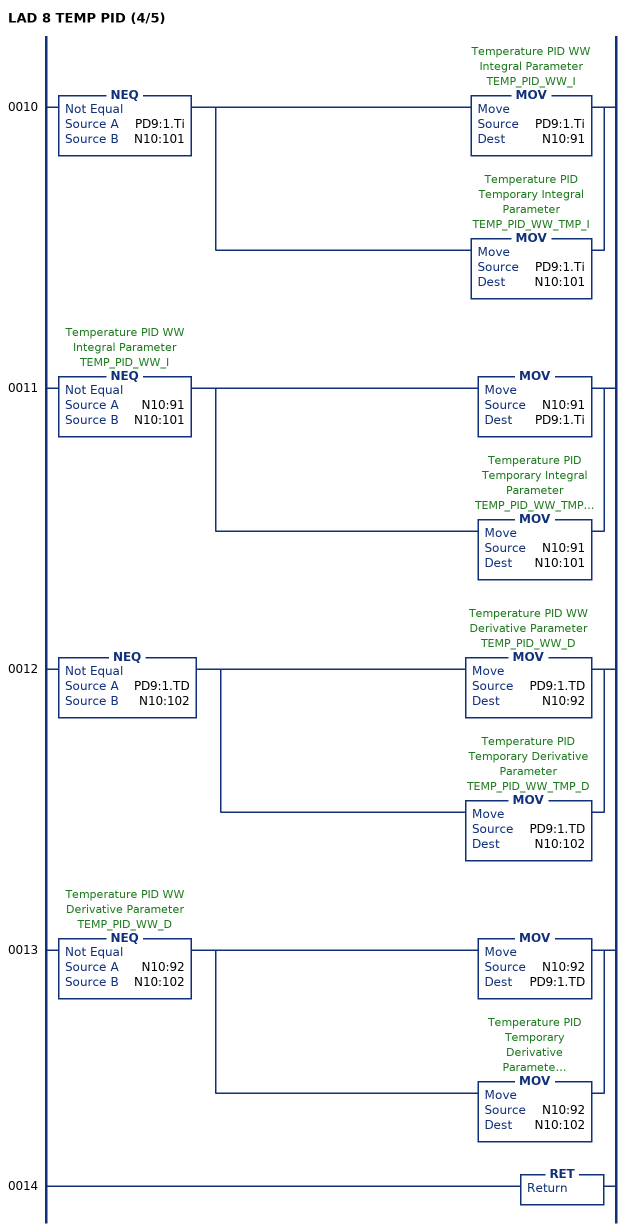
% Rung: 10 %
SOR NEQ PD9:1.Ti N10:101 BST MOV PD9:1.Ti N10:91 NXB MOV PD9:1.Ti N10:101 BND EOR
%   N10:101  TEMP_PID_WW_TMP_I  "Temperature PID Temporary Integral Parameter" %
%   N10:91  TEMP_PID_WW_I  "Temperature PID WW Integral Parameter" %
% Rung: 11 %
SOR NEQ N10:91 N10:101 BST MOV N10:91 PD9:1.Ti NXB MOV N10:91 N10:101 BND EOR
%   N10:91  TEMP_PID_WW_I  "Temperature PID WW Integral Parameter" %
%   N10:101  TEMP_PID_WW_TMP_I  "Temperature PID Temporary Integral Parameter" %
% Rung: 12 %
SOR NEQ PD9:1.TD N10:102 BST MOV PD9:1.TD N10:92 NXB MOV PD9:1.TD N10:102 BND EOR
%   N10:102  TEMP_PID_WW_TMP_D  "Temperature PID Temporary Derivative Parameter" %
%   N10:92  TEMP_PID_WW_D  "Temperature PID WW Derivative Parameter" %
% Rung: 13 %
SOR NEQ N10:92 N10:102 BST MOV N10:92 PD9:1.TD NXB MOV N10:92 N10:102 BND EOR
%   N10:92  TEMP_PID_WW_D  "Temperature PID WW Derivative Parameter" %
%   N10:102  TEMP_PID_WW_TMP_D  "Temperature PID Temporary Derivative Parameter" %
% Rung: 14 %
SOR RET EOR

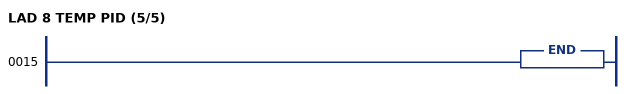
% Rung: 15 %
SOR END EOR

LADDER 9 "ANALOG OUT"
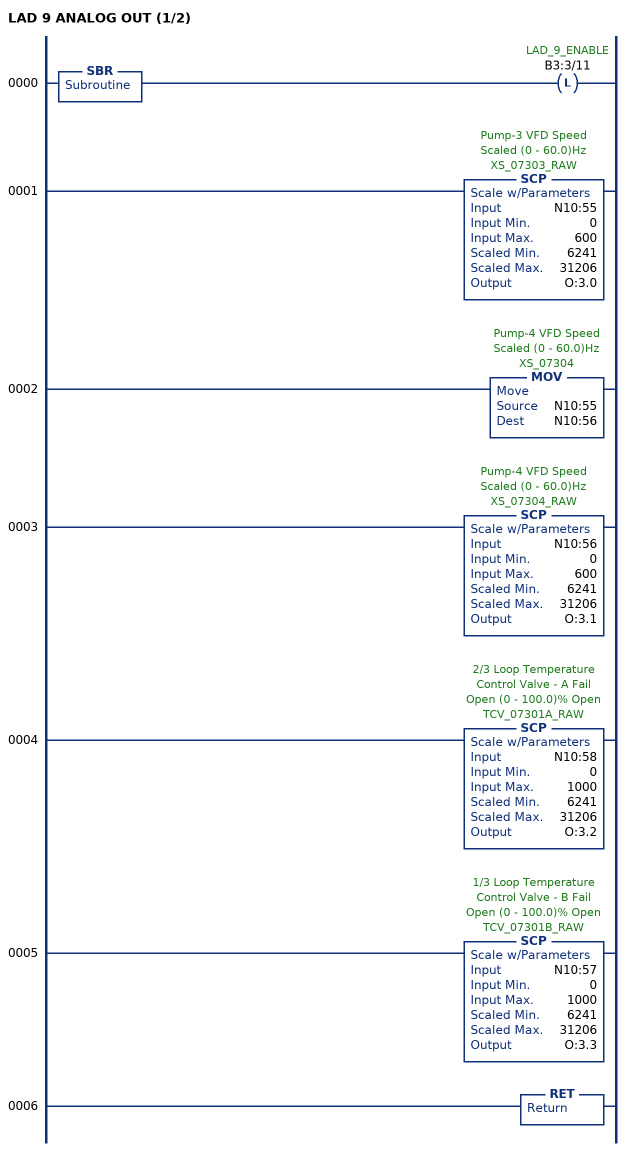
% Rung: 0 %
SOR SBR OTL B3:3/11 EOR
%   B3:3/11  LAD_9_ENABLE %
% Rung: 1 %
SOR SCP N10:55 0 600 6241 31206 O:3.0 EOR
%   N10:55  XS_07303  "Pump-3 VFD Speed Scaled (0 - 60.0)Hz" %
%   O:3.0  XS_07303_RAW  "Pump-3 VFD Speed Scaled (0 - 60.0)Hz" %
% Rung: 2 %
SOR MOV N10:55 N10:56 EOR
%   N10:55  XS_07303  "Pump-3 VFD Speed Scaled (0 - 60.0)Hz" %
%   N10:56  XS_07304  "Pump-4 VFD Speed Scaled (0 - 60.0)Hz" %
% Rung: 3 %
SOR SCP N10:56 0 600 6241 31206 O:3.1 EOR
%   N10:56  XS_07304  "Pump-4 VFD Speed Scaled (0 - 60.0)Hz" %
%   O:3.1  XS_07304_RAW  "Pump-4 VFD Speed Scaled (0 - 60.0)Hz" %
% Rung: 4 %
SOR SCP N10:58 0 1000 6241 31206 O:3.2 EOR
%   N10:58  TCV_07301B  "1/3 Loop Temperature Control Valve - B Fail Open Scaled (0 - 100.0)%" %
%   O:3.2  TCV_07301A_RAW  "2/3 Loop Temperature Control Valve - A Fail Open (0 - 100.0)% Open" %
% Rung: 5 %
SOR SCP N10:57 0 1000 6241 31206 O:3.3 EOR
%   N10:57  TCV_07301A  "2/3 Loop Temperature Control Valve - A Fail Open Scaled (0 - 100.0)%" %
%   O:3.3  TCV_07301B_RAW  "1/3 Loop Temperature Control Valve - B Fail Open (0 - 100.0)% Open" %
% Rung: 6 %
SOR RET EOR

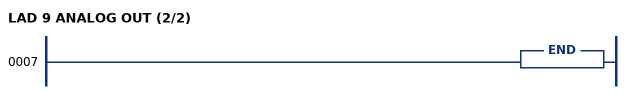
% Rung: 7 %
SOR END EOR

LADDER 10 "LCD INFO"
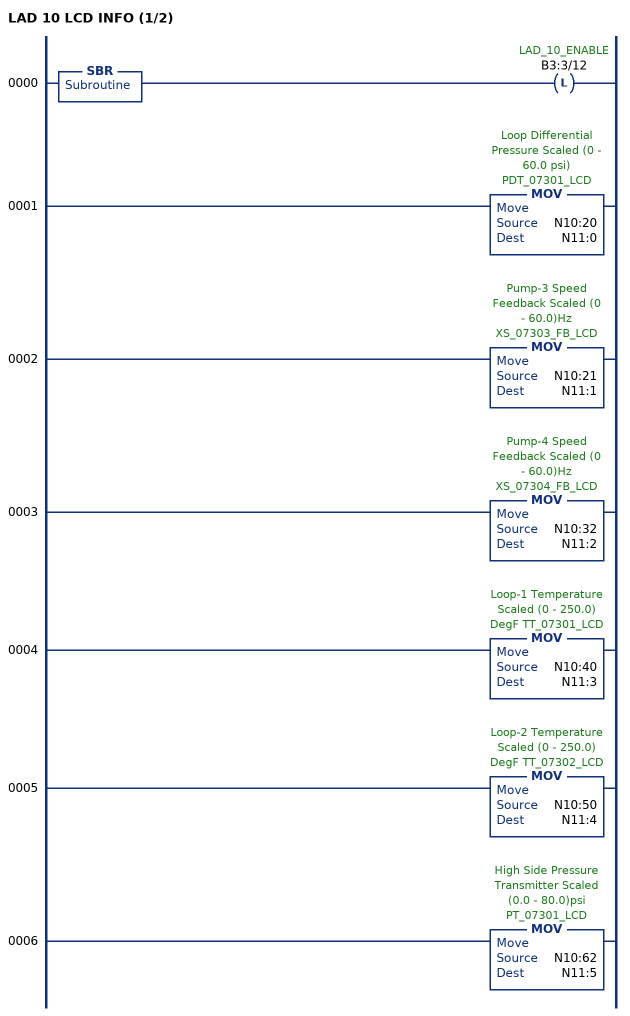
% Rung: 0 %
SOR SBR OTL B3:3/12 EOR
%   B3:3/12  LAD_10_ENABLE %
% Rung: 1 %
SOR MOV N10:20 N11:0 EOR
%   N10:20  PDT_07301  "Loop Differential Pressure Scaled (0 - 60.0 psi)" %
%   N11:0  PDT_07301_LCD  "Loop Differential Pressure Scaled (0 - 60.0 psi)" %
% Rung: 2 %
SOR MOV N10:21 N11:1 EOR
%   N10:21  XS_07303_FB  "Pump-3 Speed Feedback Scaled (0 - 60.0)Hz" %
%   N11:1  XS_07303_FB_LCD  "Pump-3 Speed Feedback Scaled (0 - 60.0)Hz" %
% Rung: 3 %
SOR MOV N10:32 N11:2 EOR
%   N10:32  XS_07304_FB  "Pump-4 Speed Feedback Scaled (0 - 60.0)Hz" %
%   N11:2  XS_07304_FB_LCD  "Pump-4 Speed Feedback Scaled (0 - 60.0)Hz" %
% Rung: 4 %
SOR MOV N10:40 N11:3 EOR
%   N10:40  TT_07301  "Loop-1 Temperature Scaled (0 - 250.0) DegF" %
%   N11:3  TT_07301_LCD  "Loop-1 Temperature Scaled (0 - 250.0) DegF" %
% Rung: 5 %
SOR MOV N10:50 N11:4 EOR
%   N10:50  TT_07302  "Loop-2 Temperature Scaled (0 - 250.0) DegF" %
%   N11:4  TT_07302_LCD  "Loop-2 Temperature Scaled (0 - 250.0) DegF" %
% Rung: 6 %
SOR MOV N10:62 N11:5 EOR
%   N10:62  PT_07301  "High Side Pressure Transmitter Scaled (0.0 - 80.0)psi" %
%   N11:5  PT_07301_LCD  "High Side Pressure Transmitter Scaled (0.0 - 80.0)psi" %

